{attribute 'qualified_only'}
{attribute 'strict'}
TYPE eOnOffState :
(
	none := 0,
	Enable := 1,
	Disable := 2
);
END_TYPE

(* stored: Version 1.1.0.1, ProductVersion 3.1.4026.18
   DUT eOnOffState: Id {3fbdbea5-7f4f-4d36-b598-d2a90ec808b6} *)
